PROGRAM PermissivesS
VAR
	AllChargeRelayClosed 	: BOOL := 0;
	AllDumpRelayOpen		: BOOL := 0;
	ReadyToCharge			: BOOL := 0;
	AllChargerEOC			: BOOL := 0;
	
	ChargerVBelowThres		: BOOL := 0;
	AllChargerHVisOFF		: BOOL := 0;
	AllChargerInhibitON		: BOOL := 0;

	AllCapsDischarged		: BOOL := 0;
	SystemIsSafe			: BOOL := 0;
END_VAR

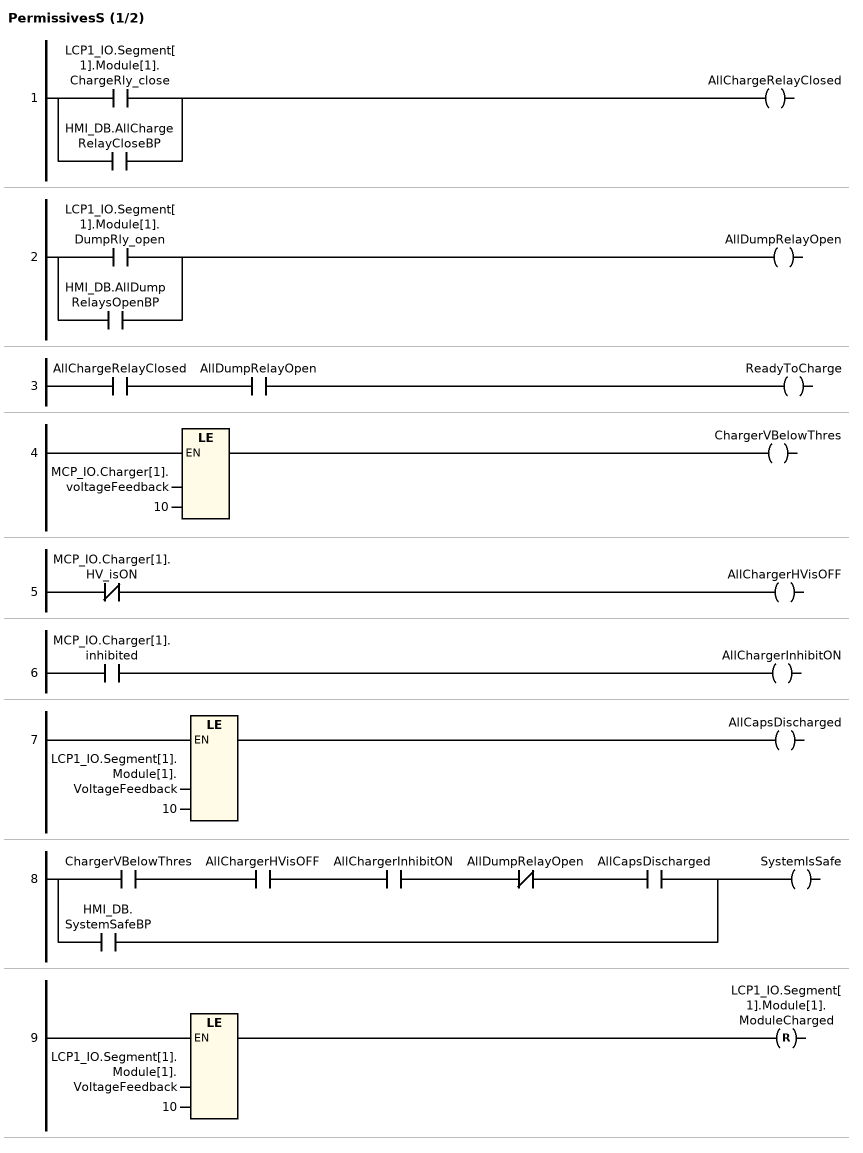
// NETWORK 1
AllChargeRelayClosed := LCP1_IO.Segment[1].Module[1].ChargeRly_close OR HMI_DB.AllChargeRelayCloseBP;

// NETWORK 2
AllDumpRelayOpen := LCP1_IO.Segment[1].Module[1].DumpRly_open OR HMI_DB.AllDumpRelaysOpenBP;

// NETWORK 3
ReadyToCharge := AllChargeRelayClosed AND AllDumpRelayOpen;

// NETWORK 4
ChargerVBelowThres := MCP_IO.Charger[1].voltageFeedback <= 10;

// NETWORK 5
AllChargerHVisOFF := NOT MCP_IO.Charger[1].HV_isON;

// NETWORK 6
AllChargerInhibitON := MCP_IO.Charger[1].inhibited;

// NETWORK 7
AllCapsDischarged := LCP1_IO.Segment[1].Module[1].VoltageFeedback <= 10;

// NETWORK 8
SystemIsSafe := ChargerVBelowThres AND AllChargerHVisOFF AND AllChargerInhibitON AND NOT AllDumpRelayOpen AND AllCapsDischarged OR HMI_DB.SystemSafeBP;

// NETWORK 9
LCP1_IO.Segment[1].Module[1].ModuleCharged R= LCP1_IO.Segment[1].Module[1].VoltageFeedback <= 10;

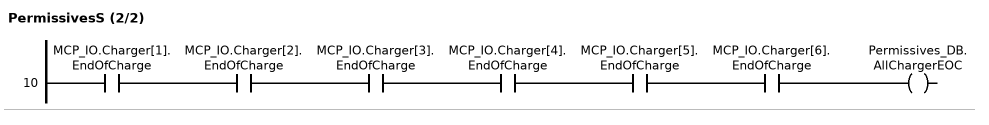
// NETWORK 10
Permissives_DB.AllChargerEOC := MCP_IO.Charger[1].EndOfCharge AND MCP_IO.Charger[2].EndOfCharge AND MCP_IO.Charger[3].EndOfCharge AND MCP_IO.Charger[4].EndOfCharge AND MCP_IO.Charger[5].EndOfCharge AND MCP_IO.Charger[6].EndOfCharge;

END_PROGRAM

(* stored: Version 1.1.0.1, ProductVersion 3.1.4024.11
   POU PermissivesS: Id {90f08704-3be2-4c8d-baf0-af04b61a9d91}, SpecialFunc None *)
